FUNCTION_BLOCK IW
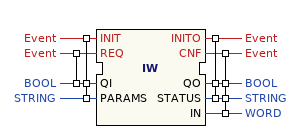
  EVENT_INPUT
    INIT WITH QI, PARAMS;
    REQ WITH QI;
  END_EVENT
  EVENT_OUTPUT
    INITO WITH QO, STATUS;
    CNF WITH QO, STATUS, IN;
  END_EVENT
  VAR_INPUT
    QI : BOOL;
    PARAMS : STRING;
  END_VAR
  VAR_OUTPUT
    QO : BOOL;
    STATUS : STRING;
    IN : WORD;
  END_VAR
END_FUNCTION_BLOCK
